TYPE E_ClientServerSteps :
(
	eUDP_STATE_IDLE		:= 0,
	eUDP_STATE_CREATE_START,
	eUDP_STATE_CREATE_WAIT,
	eUDP_STATE_SEND_START,
	eUDP_STATE_SEND_WAIT,
	eUDP_STATE_RECEIVE_START,
	eUDP_STATE_RECEIVE_WAIT,
	eUDP_STATE_CLOSE_START,
	eUDP_STATE_CLOSE_WAIT,
	eUDP_STATE_ERROR
);
END_TYPE

(* stored: Version 1.1.0.1, ProductVersion 3.1.0.20
   DUT E_ClientServerSteps: Id {f1bf31c1-7799-4639-924a-8ade29a5ca97} *)
